(* Logix 5000 project; controller Carpenter_Meter_SCP vendor 1 type 14 code 217 rev 31.11; software revision 31.01; part 4 of 7 *)
(* tags used below, declared in another part *)
   AlwaysOff : BOOL;   // Always Off Bit
   CAR100_Flowpath : BOOL;   // Carpenter MLV CAR100 Flow Path (1=OK)
   CAR100_HB_Fail : TGE_Alarm;   // Carpenter MLV CAR100 Heartbeat Fail Alarm
   CAR100_HB_Prev : DINT;   // MLV CAR100 Previous Heartbeat
   CAR100_High_Pressure_SD : BOOL;   // Carpenter MLV CAR100 High Pressure Shutdown Status
   Carpenter_ISD_Command : BOOL;   // Carpenter/Hereford ISD Command from OCC (Through Pawnee)
   Carpenter_Status_Pawnee : DINT[50];   // Carpenter Status to Pawnee
   Customer1_Pump_Status : BOOL;   // Customer #1 Pump Running Status
   Customer1_Ready_Status : BOOL;   // Customer #1 Ready Status
   FGP_ESD : TGE_Alarm;   // ESD Shutdown from FGP (HS-0020A)
   FGP_Fire_Det : TGE_Alarm;   // Fire Shutdown from FGP (YSHH-0022)
   FGP_Gas_Det : TGE_Alarm;   // Hi Gas Shutdown from FGP (ASHH-0021)
   FI_8800 : REAL;   // Meter Skid MS-8800 Flow Rate in GSV from EFM
   Hereford_Msg1 : MESSAGE;
   HRF100_Flowpath : BOOL;   // Hereford MLV HRF100 Flow Path (1=OK)
   HRF100_HB_Fail : TGE_Alarm;   // Hereford MLV HRF100 Heartbeat Fail Alarm
   HRF100_HB_Prev : DINT;   // Hereford MLV HRF100 Previous Heartbeat
   HRF100_High_Pressure_SD : BOOL;   // Hereford MLV HRF100 High Pressure Shutdown Status
   Launcher_Pig_Sig : TGE_Alarm;   // Launcher Pig Signal (ZS-1100A)
   Main_FGP_24VDC_Fail : TGE_Alarm;   // Main PLC FGP 24VDC Fail (XS-0021)
   message_timer : TIMER[10];
   MLV_CAR100_Msg1 : MESSAGE;   // Carpenter MLV (CAR100) Messaging
   MLV_CAR100_Status : DINT[50];
   MLV_HRF100_Msg1 : MESSAGE;   // Hereford MLV (HRF100) Messaging
   MLV_HRF100_Status : DINT[50];
   MS8800_Biocide_Flow_Fdbk : TGE_AI_UDT;   // Meter Skid MS-8800 Biocide Injection Rate Feedback
   MS8800_Biocide_Flow_Fdbk_AOI : TGE_AI;   // Meter Skid MS-8800 Biocide Injection Rate Feedback
   MS8800_Cust_Press : TGE_AI_UDT;   // Meter Skid MS-8800 Customer Inlet Pressure (Communicated from Cust)
   MS8800_Cust_Press_AOI : TGE_AI;   // Meter Skid MS-8800 Customer Inlet Pressure (Communicated from Cust)
   MS8800_FGP_24VDC_Fail : TGE_Alarm;   // Meter Skid MS-8800 FGP 24VDC Fail (XS-8800B)
   MS8800_Intrusion : IntrusionAlm;   // Meter Skid MS-8800 Intrusion #1 Alarm
   MS8800_PCV_Pos : TGE_AI_UDT;   // Meter Skid MS-8800 Pressure Control Valve - Position Feedback (PCV-0001)
   MS8800_PCV_Pos_AOI : TGE_AI;   // Meter Skid MS-8800 Pressure Control Valve - Position Feedback (PCV-0001)
   MS8840_Biocide_Flow_Fdbk : TGE_AI_UDT;   // Meter Skid MS-8840 Biocide Injection Rate Feedback
   MS8840_Biocide_Flow_Fdbk_AOI : TGE_AI;   // Meter Skid MS-8840 Biocide Injection Rate Feedback
   MS8840_Cust_Press : TGE_AI_UDT;   // Meter Skid MS-8840 Customer Inlet Pressure (Communicated from Cust)
   MS8840_Cust_Press_AOI : TGE_AI;   // Meter Skid MS-8840 Customer Inlet Pressure (Communicated from Cust)
   MS8840_FGP_24VDC_Fail : TGE_Alarm;   // Meter Skid MS-8840 FGP 24VDC Fail (XS-8840B)
   MS8840_Intrusion : IntrusionAlm;   // Meter Skid MS-8840 Intrusion Alarm
   MS8840_PCV_Pos : TGE_AI_UDT;   // Meter Skid MS-8840 Pressure Control Valve - Position Feedback (PCV-0041)
   MS8840_PCV_Pos_AOI : TGE_AI;   // Meter Skid MS-8840 Pressure Control Valve - Position Feedback (PCV-0041)
   one_sec_tmr : TIMER;   // One Second Pulse Timer
   Pawnee_ESD : BOOL;   // Pawnee Terminal ESD Signal (1=OK, 0 = ESD Active)
   Pawnee_Flowpath : BOOL;   // Pawnee Terminal Flow Path (1=OK)
   Pawnee_HB_Fail : TGE_Alarm;   // Pawnee Heartbeat Fail Alarm
   Pawnee_HB_Prev : DINT;   // Pawnee Heartbeat Previous Value
   Pawnee_High_Pressure_SD : BOOL;   // Pawnee High Pressure Shutdown Status
   Pawnee_Msg1 : MESSAGE;   // Pawnee Read Message
   Pawnee_Msg2 : MESSAGE;   // Pawnee Write Message
   Pawnee_OCC_HB_FAIL : BOOL;   // Pawnee OCC HB Fail
   Pawnee_Status : DINT[50];   // Pawnee Status Bits
   PDC_Bldg_Intrusion : IntrusionAlm;   // PDC Building Intrusion Alarm
   QA_Bldg_Intrusion : IntrusionAlm;   // QA Building Intrusion Alarm Bit 0-7 = Bldg Int Switch Bit 15 = Deact HS
   Sta_Stat : StaStatus;
   Station_Depart_Pig_Sig : TGE_Alarm;   // Station Departed Pig Signal (ZS-1100B)
   Station_Disch_Press : TGE_AI_UDT;   // Station Discharge Pressure - Launcher Skid (PIT-1101)
   Station_Disch_Press_AOI : TGE_AI;   // Station Discharge Pressure - Launcher Skid (PIT-1101)
   TU3000_HiHi_Lvl : TGE_Alarm;   // Sump Tank (TU-3000) Hi Hi Level Switch (LSHH-3000)
   TU3000_Leak_Detect : TGE_Alarm;   // Sump Tank (TU-3000) Leak Detected (LSH-3000)
   TU3000_Level : TGE_AI_UDT;   // Sump Tank (TU-3000) Level Transmitter (LIT-3000)
   TU3000_Level_AOI : TGE_AI;   // Sump Tank (TU-3000) Level Transmitter (LIT-3000)
   TU3100_HiHi_Lvl : TGE_Alarm;   // Sump Tank (TU-3100) Hi Hi Level Switch (LSHH-3100)
   TU3100_Leak_Detect : TGE_Alarm;   // Sump Tank (TU-3100) Leak Detected (LSH-3100)
   TU3100_Level : TGE_AI_UDT;   // Sump Tank (TU-3100) Level Transmitter (LIT-3100)
   TU3100_Level_AOI : TGE_AI;   // Sump Tank (TU-3100) Level Transmitter (LIT-3100)
   unit_msg_group : DINT;
   UPS_Fault : TGE_Alarm;   // UPS-6000 Fault (YS-6001)
   UPS_Online : TGE_Alarm;   // UPS-6000 Loss of AC Feed (YS-6000)
   watchdog_tmr : TIMER;   // Watchdog Timer for Communications
(* Communication, continued *)

ROUTINE Main_Comms   (* ladder *)
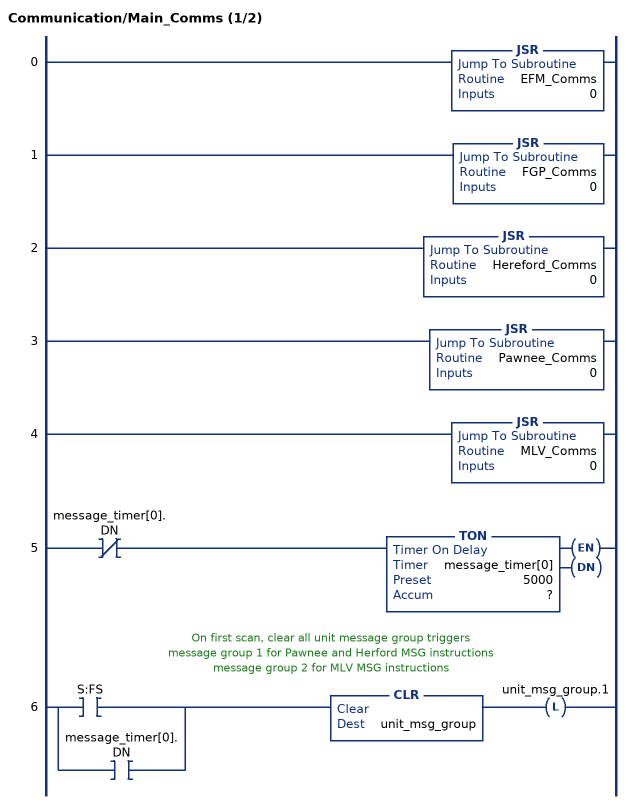
   0: JSR(EFM_Comms,0);
   1: JSR(FGP_Comms,0);
   2: JSR(Hereford_Comms,0);
   3: JSR(Pawnee_Comms,0);
   4: JSR(MLV_Comms,0);
   5: XIO(message_timer[0].DN)TON(message_timer[0],?,?);
   // On first scan, clear all unit message group triggers
   // message group 1 for Pawnee and Herford MSG instructions
   // message group 2 for MLV MSG instructions
   6: [XIC(S:FS) ,XIC(message_timer[0].DN) ]CLR(unit_msg_group)OTL(unit_msg_group.1);
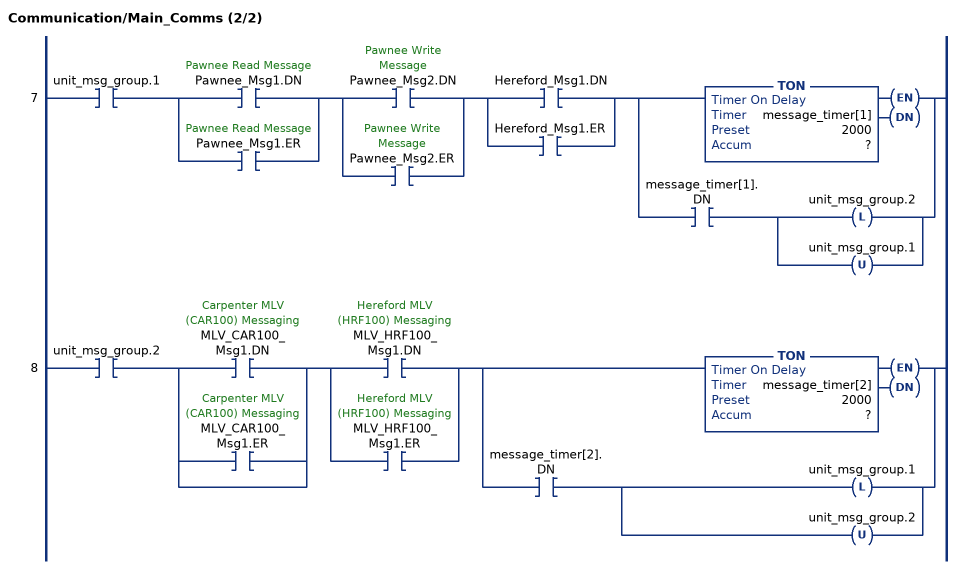
   7: XIC(unit_msg_group.1)[XIC(Pawnee_Msg1.DN) ,XIC(Pawnee_Msg1.ER) ][XIC(Pawnee_Msg2.DN) ,XIC(Pawnee_Msg2.ER) ][XIC(Hereford_Msg1.DN) ,XIC(Hereford_Msg1.ER) ][TON(message_timer[1],?,?) ,XIC(message_timer[1].DN) [OTL(unit_msg_group.2) ,OTU(unit_msg_group.1) ] ];
   8: XIC(unit_msg_group.2)[XIC(MLV_CAR100_Msg1.DN) ,XIC(MLV_CAR100_Msg1.ER) ,][XIC(MLV_HRF100_Msg1.DN) ,XIC(MLV_HRF100_Msg1.ER) ][TON(message_timer[2],?,?) ,XIC(message_timer[2].DN) [OTL(unit_msg_group.1) ,OTU(unit_msg_group.2) ] ];
END_ROUTINE

ROUTINE MLV_Comms   (* ladder *)
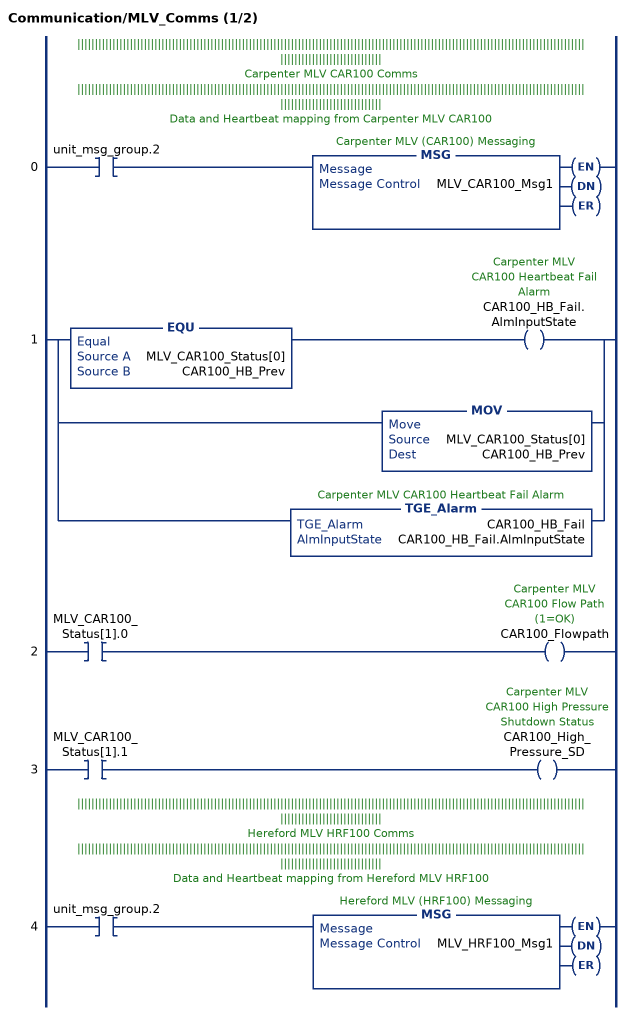
   // ||||||||||||||||||||||||||||||||||||||||||||||||||||||||||||||||||||||||||||||||||||||||||||||||||||||||||||||||||||||||||||||||||||||||||||||||||||||||||||||||||||||||||||||
   // Carpenter MLV CAR100 Comms
   // ||||||||||||||||||||||||||||||||||||||||||||||||||||||||||||||||||||||||||||||||||||||||||||||||||||||||||||||||||||||||||||||||||||||||||||||||||||||||||||||||||||||||||||||
   // Data and Heartbeat mapping from Carpenter MLV CAR100
   0: XIC(unit_msg_group.2)MSG(MLV_CAR100_Msg1);
   1: [EQU(MLV_CAR100_Status[0],CAR100_HB_Prev) OTE(CAR100_HB_Fail.AlmInputState) ,MOV(MLV_CAR100_Status[0],CAR100_HB_Prev) ,TGE_Alarm(CAR100_HB_Fail,CAR100_HB_Fail.AlmInputState) ];
   2: XIC(MLV_CAR100_Status[1].0)OTE(CAR100_Flowpath);
   3: XIC(MLV_CAR100_Status[1].1)OTE(CAR100_High_Pressure_SD);
   // ||||||||||||||||||||||||||||||||||||||||||||||||||||||||||||||||||||||||||||||||||||||||||||||||||||||||||||||||||||||||||||||||||||||||||||||||||||||||||||||||||||||||||||||
   // Hereford MLV HRF100 Comms
   // ||||||||||||||||||||||||||||||||||||||||||||||||||||||||||||||||||||||||||||||||||||||||||||||||||||||||||||||||||||||||||||||||||||||||||||||||||||||||||||||||||||||||||||||
   // Data and Heartbeat mapping from Hereford MLV HRF100
   4: XIC(unit_msg_group.2)MSG(MLV_HRF100_Msg1);
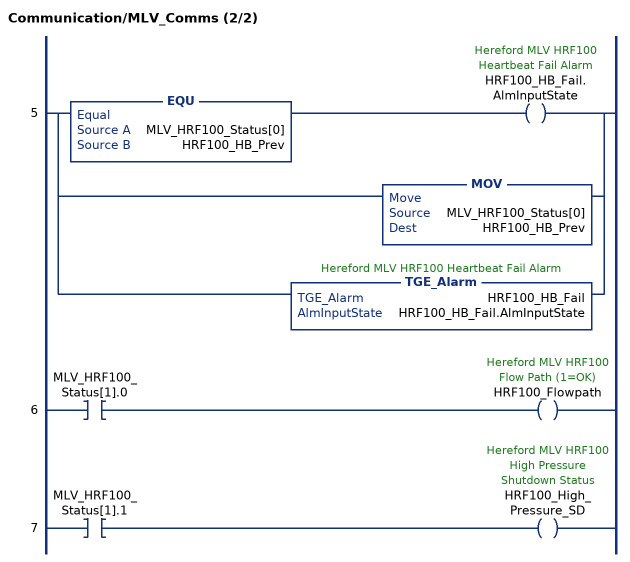
   5: [EQU(MLV_HRF100_Status[0],HRF100_HB_Prev) OTE(HRF100_HB_Fail.AlmInputState) ,MOV(MLV_HRF100_Status[0],HRF100_HB_Prev) ,TGE_Alarm(HRF100_HB_Fail,HRF100_HB_Fail.AlmInputState) ];
   6: XIC(MLV_HRF100_Status[1].0)OTE(HRF100_Flowpath);
   7: XIC(MLV_HRF100_Status[1].1)OTE(HRF100_High_Pressure_SD);
END_ROUTINE

ROUTINE Pawnee_Comms   (* ladder *)
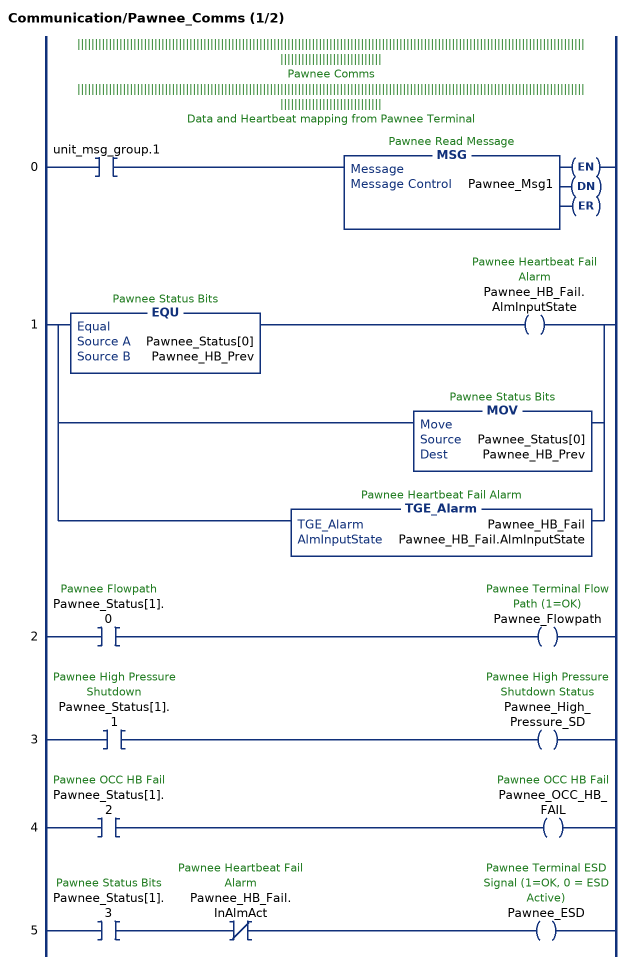
   // ||||||||||||||||||||||||||||||||||||||||||||||||||||||||||||||||||||||||||||||||||||||||||||||||||||||||||||||||||||||||||||||||||||||||||||||||||||||||||||||||||||||||||||||
   // Pawnee Comms
   // ||||||||||||||||||||||||||||||||||||||||||||||||||||||||||||||||||||||||||||||||||||||||||||||||||||||||||||||||||||||||||||||||||||||||||||||||||||||||||||||||||||||||||||||
   // Data and Heartbeat mapping from Pawnee Terminal
   0: XIC(unit_msg_group.1)MSG(Pawnee_Msg1);
   1: [EQU(Pawnee_Status[0],Pawnee_HB_Prev) OTE(Pawnee_HB_Fail.AlmInputState) ,MOV(Pawnee_Status[0],Pawnee_HB_Prev) ,TGE_Alarm(Pawnee_HB_Fail,Pawnee_HB_Fail.AlmInputState) ];
   2: XIC(Pawnee_Status[1].0)OTE(Pawnee_Flowpath);
   3: XIC(Pawnee_Status[1].1)OTE(Pawnee_High_Pressure_SD);
   4: XIC(Pawnee_Status[1].2)OTE(Pawnee_OCC_HB_FAIL);
   5: XIC(Pawnee_Status[1].3)XIO(Pawnee_HB_Fail.InAlmAct)OTE(Pawnee_ESD);
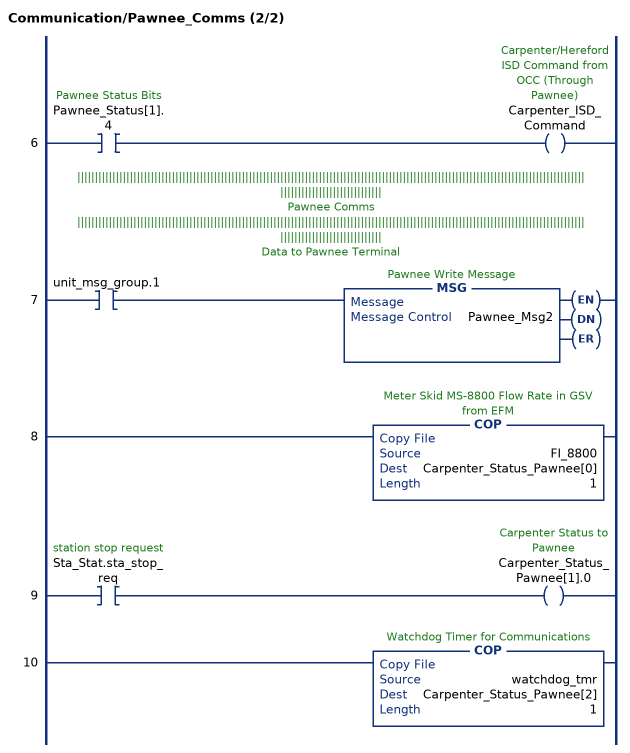
   6: XIC(Pawnee_Status[1].4)OTE(Carpenter_ISD_Command);
   // ||||||||||||||||||||||||||||||||||||||||||||||||||||||||||||||||||||||||||||||||||||||||||||||||||||||||||||||||||||||||||||||||||||||||||||||||||||||||||||||||||||||||||||||
   // Pawnee Comms
   // ||||||||||||||||||||||||||||||||||||||||||||||||||||||||||||||||||||||||||||||||||||||||||||||||||||||||||||||||||||||||||||||||||||||||||||||||||||||||||||||||||||||||||||||
   // Data to Pawnee Terminal
   7: XIC(unit_msg_group.1)MSG(Pawnee_Msg2);
   8: COP(FI_8800,Carpenter_Status_Pawnee[0],1);
   9: XIC(Sta_Stat.sta_stop_req)OTE(Carpenter_Status_Pawnee[1].0);
   10: COP(watchdog_tmr,Carpenter_Status_Pawnee[2],1);
END_ROUTINE
END_PROGRAM

PROGRAM First_Scan   (* main routine Auxiliary_Logic *)

ROUTINE Auxiliary_Logic   (* ladder *)
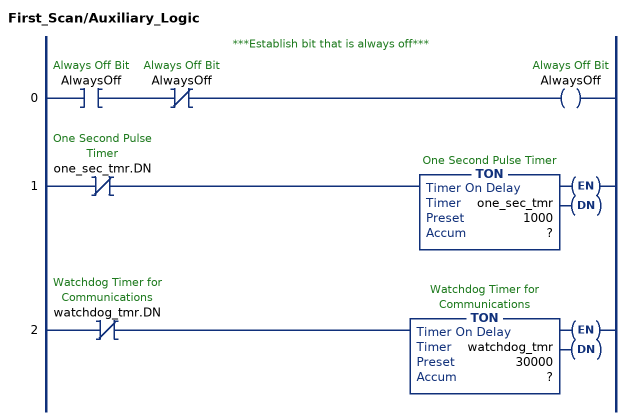
   // ***Establish bit that is always off***
   0: XIC(AlwaysOff)XIO(AlwaysOff)OTE(AlwaysOff);
   1: XIO(one_sec_tmr.DN)TON(one_sec_tmr,?,?);
   2: XIO(watchdog_tmr.DN)TON(watchdog_tmr,?,?);
END_ROUTINE
END_PROGRAM

PROGRAM Map_Inputs   (* main routine Main *)

ROUTINE Analog_Input_Map   (* ladder *)
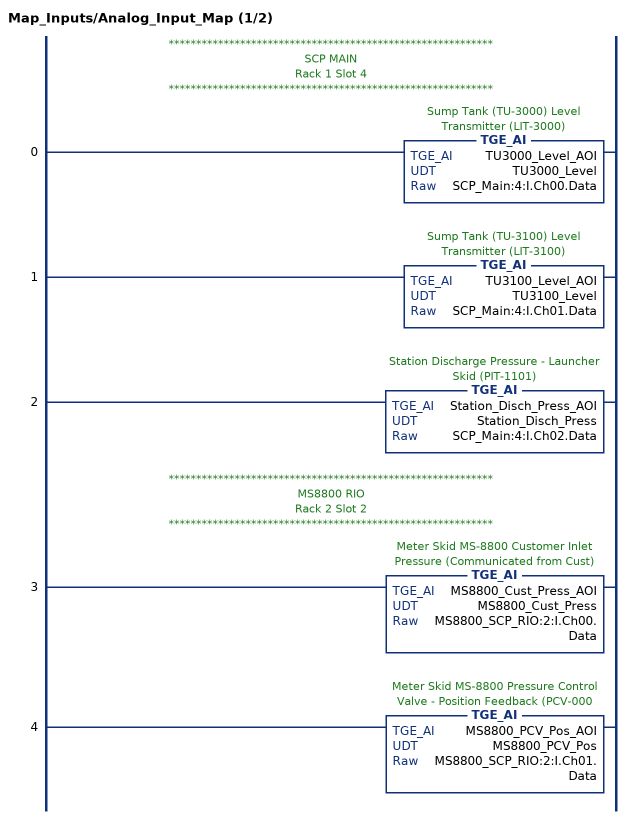
   // ***********************************************************
   // SCP MAIN
   // Rack 1 Slot 4
   // ***********************************************************
   0: TGE_AI(TU3000_Level_AOI,TU3000_Level,SCP_Main:4:I.Ch00.Data);
   1: TGE_AI(TU3100_Level_AOI,TU3100_Level,SCP_Main:4:I.Ch01.Data);
   2: TGE_AI(Station_Disch_Press_AOI,Station_Disch_Press,SCP_Main:4:I.Ch02.Data);
   // ***********************************************************
   // MS8800 RIO
   // Rack 2 Slot 2
   // ***********************************************************
   3: TGE_AI(MS8800_Cust_Press_AOI,MS8800_Cust_Press,MS8800_SCP_RIO:2:I.Ch00.Data);
   4: TGE_AI(MS8800_PCV_Pos_AOI,MS8800_PCV_Pos,MS8800_SCP_RIO:2:I.Ch01.Data);
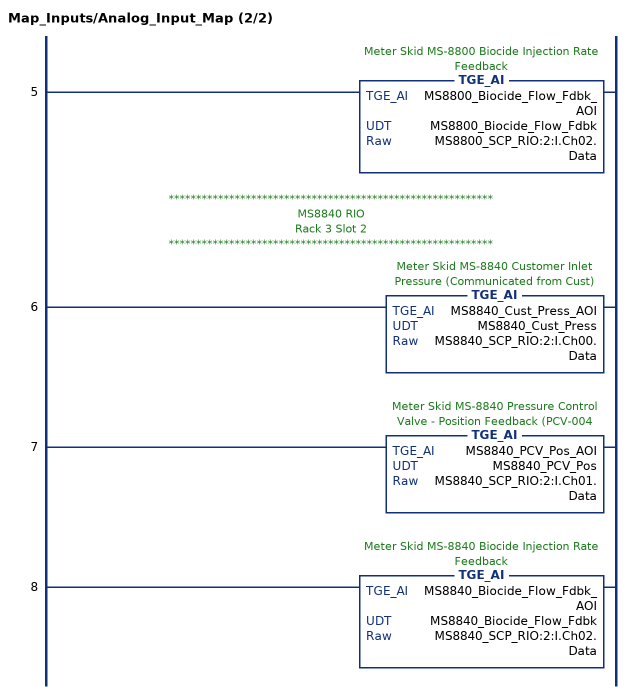
   5: TGE_AI(MS8800_Biocide_Flow_Fdbk_AOI,MS8800_Biocide_Flow_Fdbk,MS8800_SCP_RIO:2:I.Ch02.Data);
   // ***********************************************************
   // MS8840 RIO
   // Rack 3 Slot 2
   // ***********************************************************
   6: TGE_AI(MS8840_Cust_Press_AOI,MS8840_Cust_Press,MS8840_SCP_RIO:2:I.Ch00.Data);
   7: TGE_AI(MS8840_PCV_Pos_AOI,MS8840_PCV_Pos,MS8840_SCP_RIO:2:I.Ch01.Data);
   8: TGE_AI(MS8840_Biocide_Flow_Fdbk_AOI,MS8840_Biocide_Flow_Fdbk,MS8840_SCP_RIO:2:I.Ch02.Data);
END_ROUTINE

ROUTINE Discrete_Input_Map   (* ladder *)
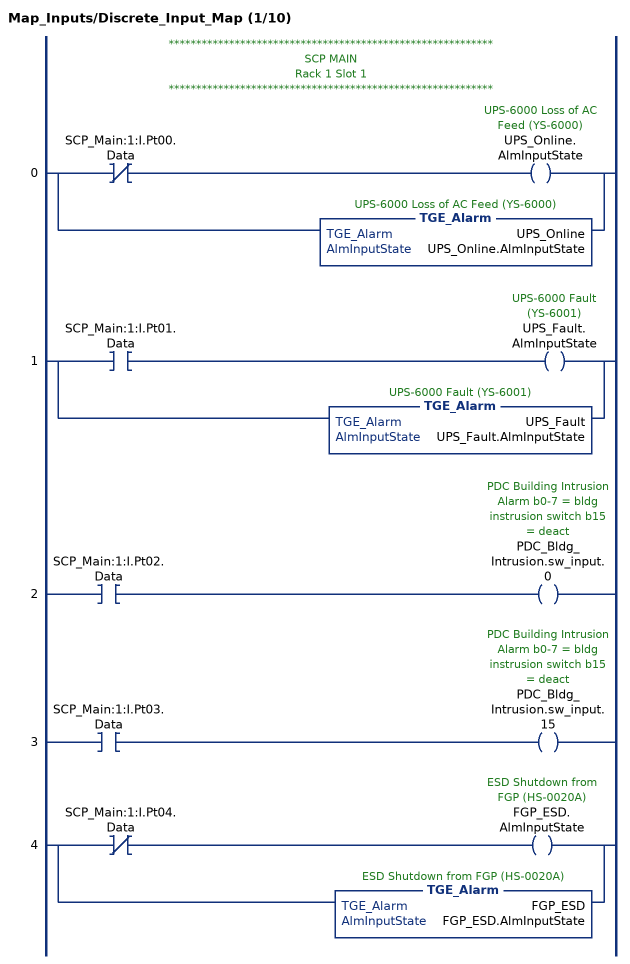
   // ***********************************************************
   // SCP MAIN
   // Rack 1 Slot 1
   // ***********************************************************
   0: [XIO(SCP_Main:1:I.Pt00.Data) OTE(UPS_Online.AlmInputState) ,TGE_Alarm(UPS_Online,UPS_Online.AlmInputState) ];
   1: [XIC(SCP_Main:1:I.Pt01.Data) OTE(UPS_Fault.AlmInputState) ,TGE_Alarm(UPS_Fault,UPS_Fault.AlmInputState) ];
   2: XIC(SCP_Main:1:I.Pt02.Data)OTE(PDC_Bldg_Intrusion.sw_input.0);
   3: XIC(SCP_Main:1:I.Pt03.Data)OTE(PDC_Bldg_Intrusion.sw_input.15);
   4: [XIO(SCP_Main:1:I.Pt04.Data) OTE(FGP_ESD.AlmInputState) ,TGE_Alarm(FGP_ESD,FGP_ESD.AlmInputState) ];
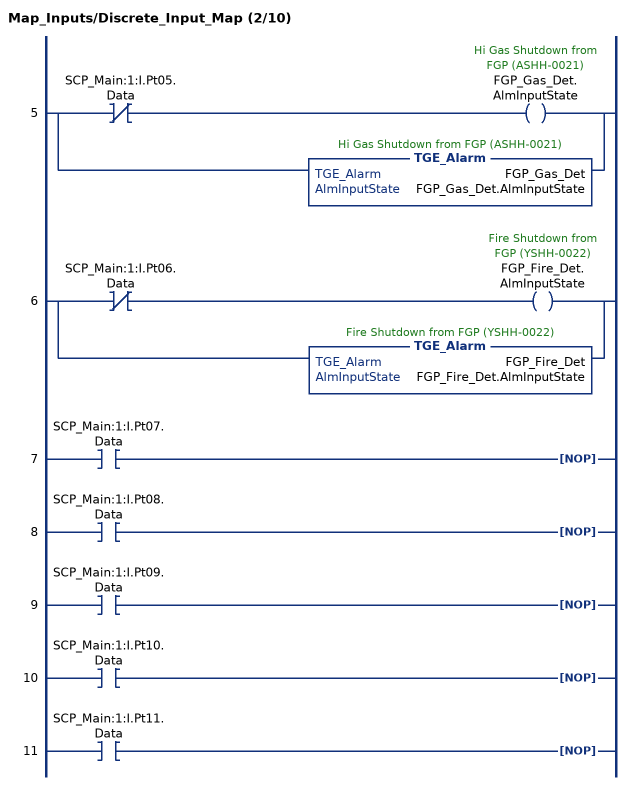
   5: [XIO(SCP_Main:1:I.Pt05.Data) OTE(FGP_Gas_Det.AlmInputState) ,TGE_Alarm(FGP_Gas_Det,FGP_Gas_Det.AlmInputState) ];
   6: [XIO(SCP_Main:1:I.Pt06.Data) OTE(FGP_Fire_Det.AlmInputState) ,TGE_Alarm(FGP_Fire_Det,FGP_Fire_Det.AlmInputState) ];
   7: XIC(SCP_Main:1:I.Pt07.Data)NOP();
   8: XIC(SCP_Main:1:I.Pt08.Data)NOP();
   9: XIC(SCP_Main:1:I.Pt09.Data)NOP();
   10: XIC(SCP_Main:1:I.Pt10.Data)NOP();
   11: XIC(SCP_Main:1:I.Pt11.Data)NOP();
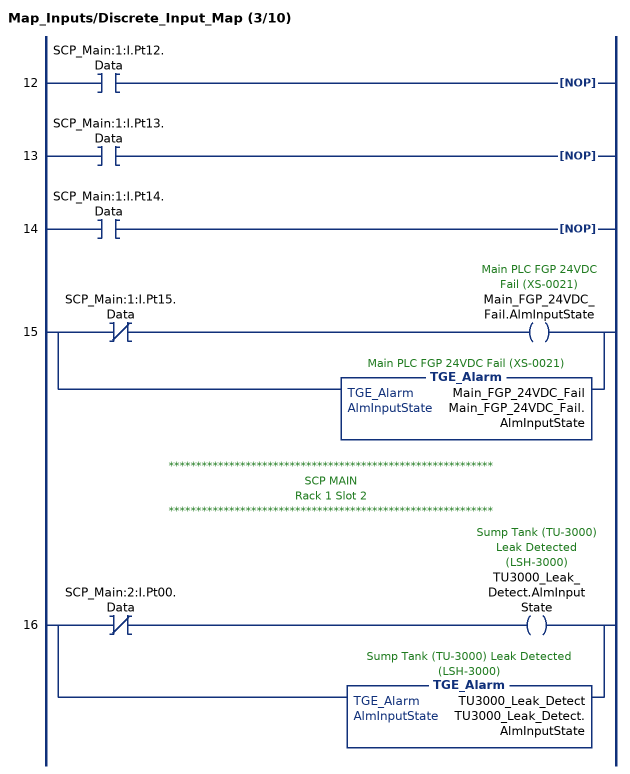
   12: XIC(SCP_Main:1:I.Pt12.Data)NOP();
   13: XIC(SCP_Main:1:I.Pt13.Data)NOP();
   14: XIC(SCP_Main:1:I.Pt14.Data)NOP();
   15: [XIO(SCP_Main:1:I.Pt15.Data) OTE(Main_FGP_24VDC_Fail.AlmInputState) ,TGE_Alarm(Main_FGP_24VDC_Fail,Main_FGP_24VDC_Fail.AlmInputState) ];
   // ***********************************************************
   // SCP MAIN
   // Rack 1 Slot 2
   // ***********************************************************
   16: [XIO(SCP_Main:2:I.Pt00.Data) OTE(TU3000_Leak_Detect.AlmInputState) ,TGE_Alarm(TU3000_Leak_Detect,TU3000_Leak_Detect.AlmInputState) ];
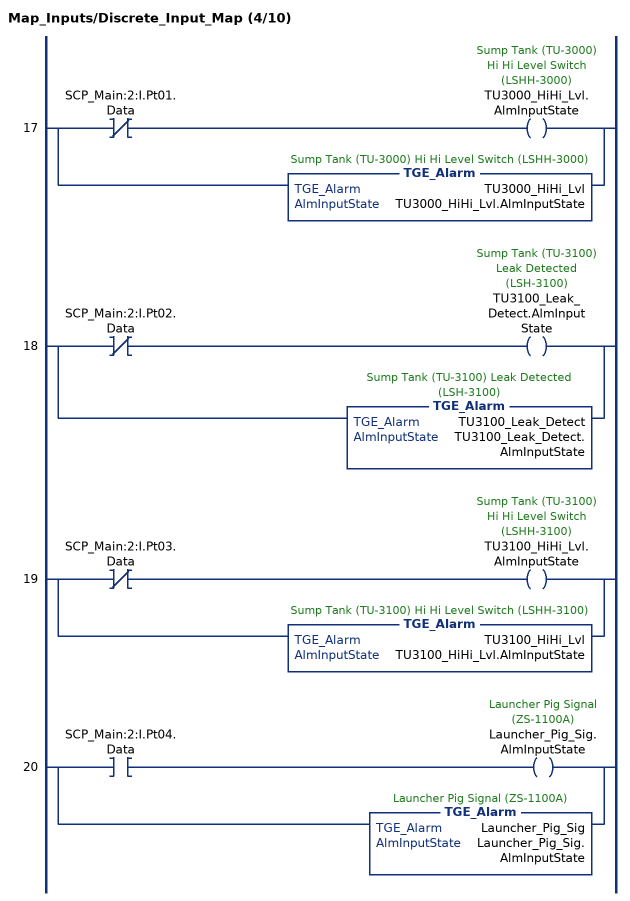
   17: [XIO(SCP_Main:2:I.Pt01.Data) OTE(TU3000_HiHi_Lvl.AlmInputState) ,TGE_Alarm(TU3000_HiHi_Lvl,TU3000_HiHi_Lvl.AlmInputState) ];
   18: [XIO(SCP_Main:2:I.Pt02.Data) OTE(TU3100_Leak_Detect.AlmInputState) ,TGE_Alarm(TU3100_Leak_Detect,TU3100_Leak_Detect.AlmInputState) ];
   19: [XIO(SCP_Main:2:I.Pt03.Data) OTE(TU3100_HiHi_Lvl.AlmInputState) ,TGE_Alarm(TU3100_HiHi_Lvl,TU3100_HiHi_Lvl.AlmInputState) ];
   20: [XIC(SCP_Main:2:I.Pt04.Data) OTE(Launcher_Pig_Sig.AlmInputState) ,TGE_Alarm(Launcher_Pig_Sig,Launcher_Pig_Sig.AlmInputState) ];
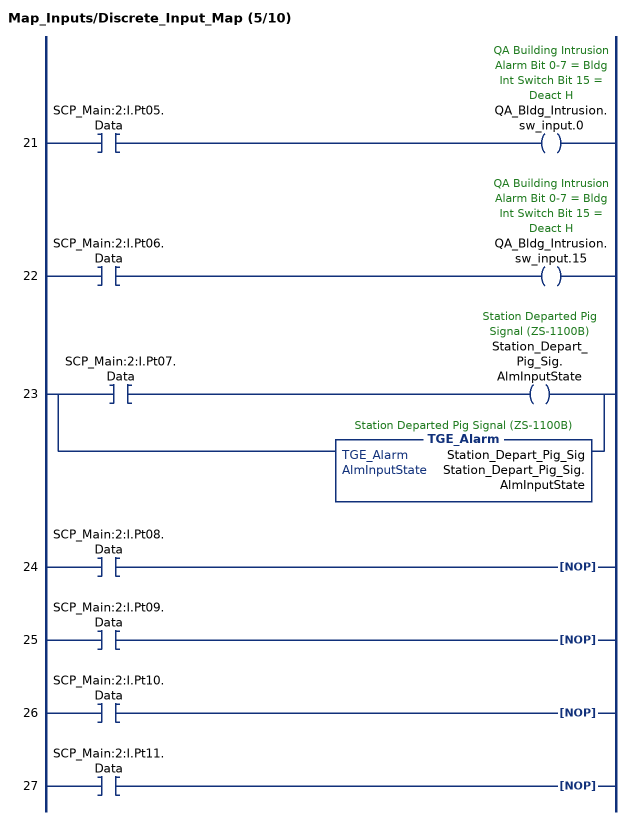
   21: XIC(SCP_Main:2:I.Pt05.Data)OTE(QA_Bldg_Intrusion.sw_input.0);
   22: XIC(SCP_Main:2:I.Pt06.Data)OTE(QA_Bldg_Intrusion.sw_input.15);
   23: [XIC(SCP_Main:2:I.Pt07.Data) OTE(Station_Depart_Pig_Sig.AlmInputState) ,TGE_Alarm(Station_Depart_Pig_Sig,Station_Depart_Pig_Sig.AlmInputState) ];
   24: XIC(SCP_Main:2:I.Pt08.Data)NOP();
   25: XIC(SCP_Main:2:I.Pt09.Data)NOP();
   26: XIC(SCP_Main:2:I.Pt10.Data)NOP();
   27: XIC(SCP_Main:2:I.Pt11.Data)NOP();
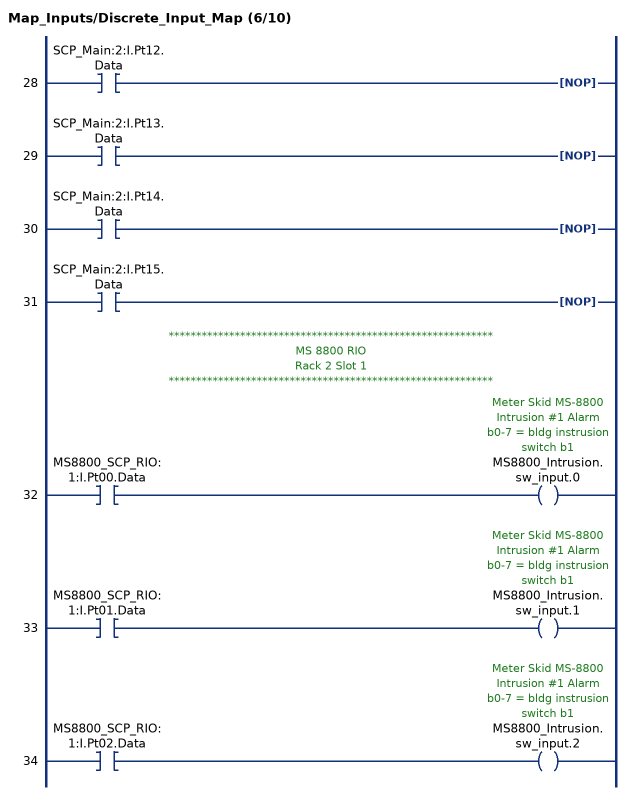
   28: XIC(SCP_Main:2:I.Pt12.Data)NOP();
   29: XIC(SCP_Main:2:I.Pt13.Data)NOP();
   30: XIC(SCP_Main:2:I.Pt14.Data)NOP();
   31: XIC(SCP_Main:2:I.Pt15.Data)NOP();
   // ***********************************************************
   // MS 8800 RIO
   // Rack 2 Slot 1
   // ***********************************************************
   32: XIC(MS8800_SCP_RIO:1:I.Pt00.Data)OTE(MS8800_Intrusion.sw_input.0);
   33: XIC(MS8800_SCP_RIO:1:I.Pt01.Data)OTE(MS8800_Intrusion.sw_input.1);
   34: XIC(MS8800_SCP_RIO:1:I.Pt02.Data)OTE(MS8800_Intrusion.sw_input.2);
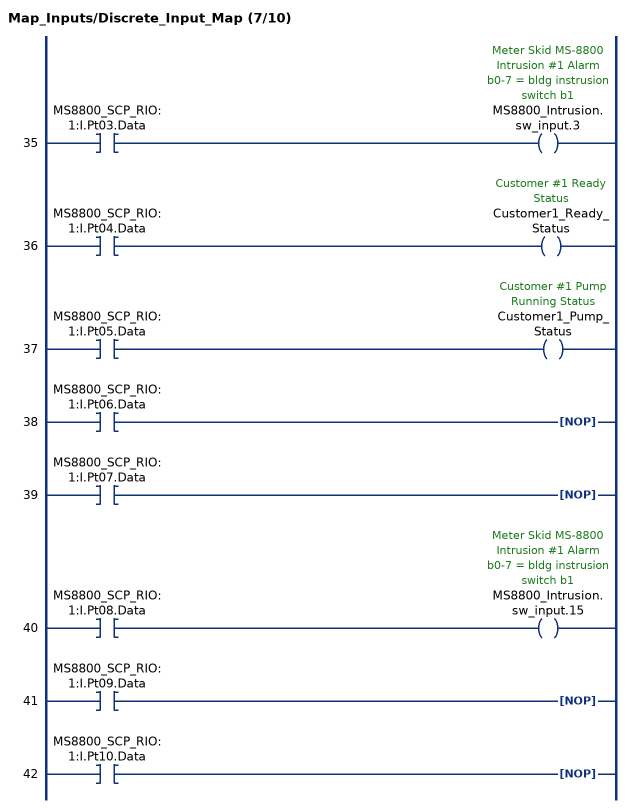
   35: XIC(MS8800_SCP_RIO:1:I.Pt03.Data)OTE(MS8800_Intrusion.sw_input.3);
   36: XIC(MS8800_SCP_RIO:1:I.Pt04.Data)OTE(Customer1_Ready_Status);
   37: XIC(MS8800_SCP_RIO:1:I.Pt05.Data)OTE(Customer1_Pump_Status);
   38: XIC(MS8800_SCP_RIO:1:I.Pt06.Data)NOP();
   39: XIC(MS8800_SCP_RIO:1:I.Pt07.Data)NOP();
   40: XIC(MS8800_SCP_RIO:1:I.Pt08.Data)OTE(MS8800_Intrusion.sw_input.15);
   41: XIC(MS8800_SCP_RIO:1:I.Pt09.Data)NOP();
   42: XIC(MS8800_SCP_RIO:1:I.Pt10.Data)NOP();
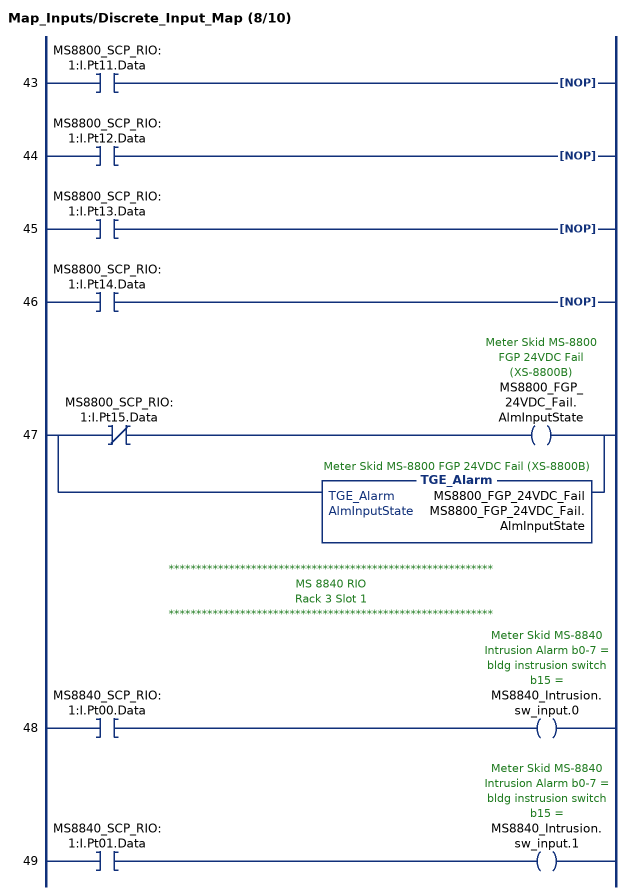
   43: XIC(MS8800_SCP_RIO:1:I.Pt11.Data)NOP();
   44: XIC(MS8800_SCP_RIO:1:I.Pt12.Data)NOP();
   45: XIC(MS8800_SCP_RIO:1:I.Pt13.Data)NOP();
   46: XIC(MS8800_SCP_RIO:1:I.Pt14.Data)NOP();
   47: [XIO(MS8800_SCP_RIO:1:I.Pt15.Data) OTE(MS8800_FGP_24VDC_Fail.AlmInputState) ,TGE_Alarm(MS8800_FGP_24VDC_Fail,MS8800_FGP_24VDC_Fail.AlmInputState) ];
   // ***********************************************************
   // MS 8840 RIO
   // Rack 3 Slot 1
   // ***********************************************************
   48: XIC(MS8840_SCP_RIO:1:I.Pt00.Data)OTE(MS8840_Intrusion.sw_input.0);
   49: XIC(MS8840_SCP_RIO:1:I.Pt01.Data)OTE(MS8840_Intrusion.sw_input.1);
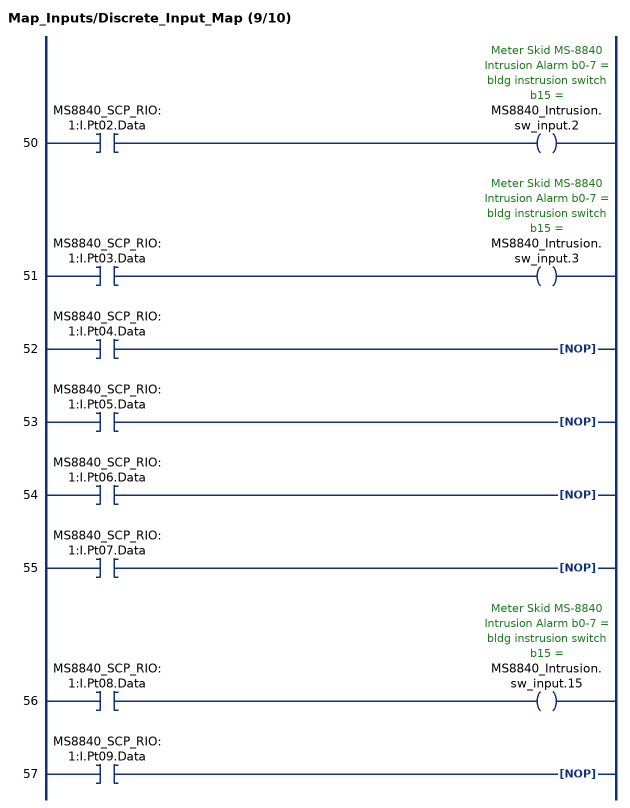
   50: XIC(MS8840_SCP_RIO:1:I.Pt02.Data)OTE(MS8840_Intrusion.sw_input.2);
   51: XIC(MS8840_SCP_RIO:1:I.Pt03.Data)OTE(MS8840_Intrusion.sw_input.3);
   52: XIC(MS8840_SCP_RIO:1:I.Pt04.Data)NOP();
   53: XIC(MS8840_SCP_RIO:1:I.Pt05.Data)NOP();
   54: XIC(MS8840_SCP_RIO:1:I.Pt06.Data)NOP();
   55: XIC(MS8840_SCP_RIO:1:I.Pt07.Data)NOP();
   56: XIC(MS8840_SCP_RIO:1:I.Pt08.Data)OTE(MS8840_Intrusion.sw_input.15);
   57: XIC(MS8840_SCP_RIO:1:I.Pt09.Data)NOP();
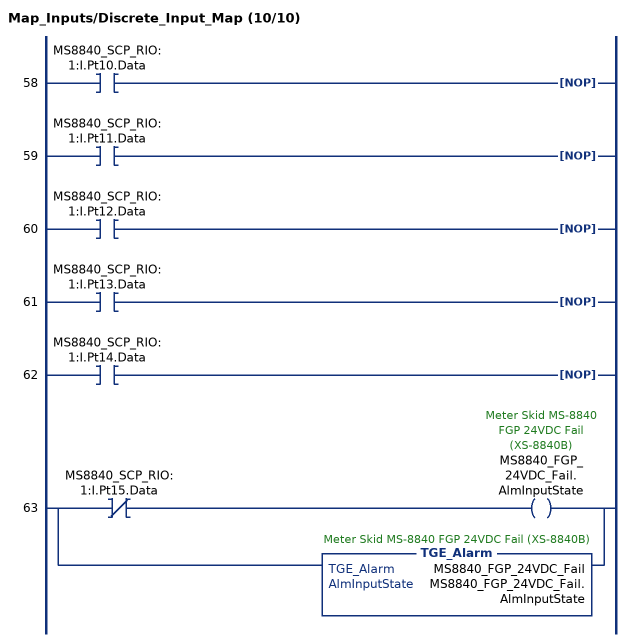
   58: XIC(MS8840_SCP_RIO:1:I.Pt10.Data)NOP();
   59: XIC(MS8840_SCP_RIO:1:I.Pt11.Data)NOP();
   60: XIC(MS8840_SCP_RIO:1:I.Pt12.Data)NOP();
   61: XIC(MS8840_SCP_RIO:1:I.Pt13.Data)NOP();
   62: XIC(MS8840_SCP_RIO:1:I.Pt14.Data)NOP();
   63: [XIO(MS8840_SCP_RIO:1:I.Pt15.Data) OTE(MS8840_FGP_24VDC_Fail.AlmInputState) ,TGE_Alarm(MS8840_FGP_24VDC_Fail,MS8840_FGP_24VDC_Fail.AlmInputState) ];
END_ROUTINE
